TYPE CellDataBlock :
UNION
	reserved : ARRAY[1..64] OF WORD; //memeory occupation
	axis : commAxis;
	cylinder : commCylinder;
	signal : commSignal;
	command : commCommandGeneric;
	unit : commUnitGeneric;
	//----------
	//	New added , 20191228
	//----------
	vacuum : commVacuum;
END_UNION
END_TYPE

(* stored: Version 1.1.0.1, ProductVersion 3.1.4024.0
   DUT CellDataBlock: Id {45a09079-c4b6-4675-89db-e70c1695c394} *)
